(* PLC project Ben_Harrison_Prototype, Beckhoff Automation GmbH TwinCAT PLC Control 3.5.13.21 *)
(* stored: creationDateTime 2024-01-25T14:00:56.1741146, modificationDateTime 2024-01-25T14:00:56.1828941 *)

INTERFACE I_Disposable
METHOD Dispose
VAR_INPUT
END_VAR
END_METHOD
END_INTERFACE

INTERFACE I_DrawableShape EXTENDS I_Disposable
METHOD Clone : I_DrawableShape
VAR_INPUT
END_VAR
END_METHOD
METHOD Draw
VAR_INPUT
END_VAR
END_METHOD
END_INTERFACE

{attribute 'enable_dynamic_creation'}
FUNCTION_BLOCK Circle EXTENDS Disposable IMPLEMENTS I_DrawableShape
VAR
	_radius: INT;
END_VAR

                  
                

METHOD Clone : I_DrawableShape
VAR
	pCircle : POINTER TO Circle;	
END_VAR
                        pCircle := __NEW(Circle);
pCircle^.radius := radius;
Clone := pCircle^;
                      
END_METHOD

METHOD Draw

VAR
	str : STRING;
END_VAR
                        str := TO_STRING(radius);
ADSLOGSTR(msgCtrlMask :=ADSLOG_MSGTYPE_HINT, msgFmtStr :='Draw circle with radius: %s', strArg := str);
                      
END_METHOD

PROPERTY Radius : INT
GET
VAR
END_VAR
                          Radius := _radius;
                        
END_GET
SET
VAR
END_VAR
                          _radius := Radius;
                        
END_SET
END_PROPERTY
END_FUNCTION_BLOCK

FUNCTION_BLOCK Disposable
VAR
END_VAR

                  
                

METHOD PUBLIC Dispose
VAR_INPUT
END_VAR
                        __DELETE(THIS);
                      
END_METHOD
END_FUNCTION_BLOCK

{attribute 'enable_dynamic_creation'}
FUNCTION_BLOCK Rectangle EXTENDS Disposable IMPLEMENTS I_DrawableShape
VAR
	_width: INT;
    _height: INT;
END_VAR

                  
                

METHOD Clone : I_DrawableShape
VAR
	pRectangle : POINTER TO Rectangle;
END_VAR
                        pRectangle := __NEW(Rectangle);
pRectangle^.Width := Width;
pRectangle^.Height := Height;
Clone := pRectangle^;
                      
END_METHOD

METHOD Draw
VAR
	str_width : STRING;
	str_height : STRING;
	str : STRING;
END_VAR
                        str_width := CONCAT(STR1 := 'width: ', STR2 := TO_STRING(Width));
str_height := CONCAT(STR1 := 'height: ', STR2 := TO_STRING(Height));
str := CONCAT(STR1 := str_width, STR2 := str_height);
ADSLOGSTR(msgCtrlMask := ADSLOG_MSGTYPE_HINT, msgFmtStr := 'Draw Rectangle with:  %s', strArg := str);
                      
END_METHOD

PROPERTY PUBLIC Height : INT
GET
VAR
END_VAR
                          Height := _height;
                        
END_GET
SET
PUBLIC 
VAR
END_VAR
                          _height := Height;
                        
END_SET
END_PROPERTY

PROPERTY PUBLIC Width : INT
GET
VAR
END_VAR
                          Width := _width;
                        
END_GET
SET
PUBLIC 
VAR
END_VAR
                          _width := Width;
                        
END_SET
END_PROPERTY
END_FUNCTION_BLOCK

PROGRAM MAIN
VAR
    originalRectangle: Rectangle;
    clonedRectangle: I_DrawableShape;
	
    originalCircle: Circle;
    clonedCircle: I_DrawableShape;
	
	bRequest : BOOL;
	counter: INT;

END_VAR

                  // https://refactoring.guru/design-patterns/prototype

// Recuerda que el patrón Prototipo permite crear nuevos objetos clonando un objeto existente, evitando así la necesidad de crear nuevas instancias desde cero.

// porque salen varios mensajes:
// https://github.com/tcunit/TcUnit/issues/92
// solución temporal : Unload project...
IF bRequest THEN
	
	// rectangle example 
	originalRectangle.Width := 10;
	originalRectangle.Height := 5;
	originalRectangle.Draw();
	clonedRectangle := originalRectangle.clone();
	clonedRectangle.Draw();
	clonedRectangle.Dispose(); 
	
	// circle example 
	originalCircle.Radius := 7;
	originalCircle.Draw();
	clonedCircle := originalCircle.clone();
	clonedCircle.Draw();
	clonedCircle.Dispose(); 
	
	// report request info
	bRequest := FALSE;
	counter := counter + 1;
	ADSLOGSTR(msgCtrlMask :=ADSLOG_MSGTYPE_HINT, msgFmtStr :='test: %s', strArg := TO_STRING(counter));

END_IF
                
END_PROGRAM

CONFIGURATION Application
  RESOURCE Ben_Harrison_Prototype ON PLC
    TASK PlcTask(INTERVAL := T#0ms, PRIORITY := 20);
    PROGRAM MAIN WITH PlcTask : MAIN;
  END_RESOURCE
END_CONFIGURATION
